(* IEC 61131-3 sources: TeoriaDeControl-NodeMCU/Lab2/build, 2 files *)

(* ---- plc.st ---- *)
TYPE
  LOGLEVEL : (CRITICAL, WARNING, INFO, DEBUG) := INFO;
END_TYPE

FUNCTION_BLOCK LOGGER
  VAR_INPUT
    TRIG : BOOL;
    MSG : STRING;
    LEVEL : LOGLEVEL := INFO;
  END_VAR
  VAR
    TRIG0 : BOOL;
  END_VAR

  IF TRIG AND NOT TRIG0 THEN
  {{
   LogMessage(GetFbVar(LEVEL),(char*)GetFbVar(MSG, .body),GetFbVar(MSG, .len));
  }}
  END_IF;
  TRIG0:=TRIG;
END_FUNCTION_BLOCK

FUNCTION_BLOCK python_eval
  VAR_INPUT
    TRIG : BOOL;
    CODE : STRING;
  END_VAR
  VAR_OUTPUT
    ACK : BOOL;
    RESULT : STRING;
  END_VAR
  VAR
    STATE : DWORD;
    BUFFER : STRING;
    PREBUFFER : STRING;
    TRIGM1 : BOOL;
    TRIGGED : BOOL;
  END_VAR

  {extern void __PythonEvalFB(int, PYTHON_EVAL*);__PythonEvalFB(0, data__);}
END_FUNCTION_BLOCK

FUNCTION_BLOCK python_poll
  VAR_INPUT
    TRIG : BOOL;
    CODE : STRING;
  END_VAR
  VAR_OUTPUT
    ACK : BOOL;
    RESULT : STRING;
  END_VAR
  VAR
    STATE : DWORD;
    BUFFER : STRING;
    PREBUFFER : STRING;
    TRIGM1 : BOOL;
    TRIGGED : BOOL;
  END_VAR

  {extern void __PythonEvalFB(int, PYTHON_EVAL*);__PythonEvalFB(1,(PYTHON_EVAL*)(void*)data__);}
END_FUNCTION_BLOCK

FUNCTION_BLOCK python_gear
  VAR_INPUT
    N : UINT;
    TRIG : BOOL;
    CODE : STRING;
  END_VAR
  VAR_OUTPUT
    ACK : BOOL;
    RESULT : STRING;
  END_VAR
  VAR
    py_eval : python_eval;
    COUNTER : UINT;
    _TMP_ADD10_OUT : UINT;
    _TMP_EQ13_OUT : BOOL;
    _TMP_SEL15_OUT : UINT;
    _TMP_AND7_OUT : BOOL;
  END_VAR

  _TMP_ADD10_OUT := ADD(COUNTER, 1);
  _TMP_EQ13_OUT := EQ(N, _TMP_ADD10_OUT);
  _TMP_SEL15_OUT := SEL(_TMP_EQ13_OUT, _TMP_ADD10_OUT, 0);
  COUNTER := _TMP_SEL15_OUT;
  _TMP_AND7_OUT := AND(_TMP_EQ13_OUT, TRIG);
  py_eval(TRIG := _TMP_AND7_OUT, CODE := CODE);
  ACK := py_eval.ACK;
  RESULT := py_eval.RESULT;
END_FUNCTION_BLOCK

PROGRAM Lab2
  VAR
    micro : INT;
    led1 : BOOL := 0;
    led2 : BOOL := 0;
    led3 : BOOL := 0;
    rele : BOOL := 0;
  END_VAR
  VAR
    TP1 : TP;
    TP2 : TP;
    TP3 : TP;
    TP4 : TP;
    _TMP_LE14_OUT : BOOL;
    _TMP_LE3_OUT : BOOL;
    _TMP_LE6_OUT : BOOL;
  END_VAR

  _TMP_LE14_OUT := LE(micro, 600);
  TP1(IN := _TMP_LE14_OUT, PT := T#10s);
  rele := TP1.Q;
  TP3(IN := _TMP_LE14_OUT, PT := T#3s);
  led3 := TP3.Q;
  _TMP_LE3_OUT := LE(micro, 800);
  TP2(IN := _TMP_LE3_OUT, PT := T#6s);
  led2 := TP2.Q;
  _TMP_LE6_OUT := LE(micro, 1000);
  TP4(IN := _TMP_LE6_OUT, PT := T#9s);
  led1 := TP4.Q;
END_PROGRAM

CONFIGURATION Config0

  RESOURCE Res0 ON PLC
    TASK task0(INTERVAL := T#20ms,PRIORITY := 0);
    PROGRAM instance0 WITH task0 : Lab2;
  END_RESOURCE
END_CONFIGURATION

(* ---- generated_plc.st ---- *)
PROGRAM Lab2
  VAR
    micro AT %IW0 : INT;
    led1 AT %QX0.1 : BOOL := 0;
    led2 AT %QX0.2 : BOOL := 0;
    led3 AT %QX0.3 : BOOL := 0;
    rele AT %QX0.0 : BOOL := 0;
  END_VAR
  VAR
    TP1 : TP;
    TP2 : TP;
    TP3 : TP;
    TP4 : TP;
    _TMP_LE14_OUT : BOOL;
    _TMP_LE3_OUT : BOOL;
    _TMP_LE6_OUT : BOOL;
  END_VAR

  _TMP_LE14_OUT := LE(micro, 600);
  TP1(IN := _TMP_LE14_OUT, PT := T#10s);
  rele := TP1.Q;
  TP3(IN := _TMP_LE14_OUT, PT := T#3s);
  led3 := TP3.Q;
  _TMP_LE3_OUT := LE(micro, 800);
  TP2(IN := _TMP_LE3_OUT, PT := T#6s);
  led2 := TP2.Q;
  _TMP_LE6_OUT := LE(micro, 1000);
  TP4(IN := _TMP_LE6_OUT, PT := T#9s);
  led1 := TP4.Q;
END_PROGRAM

CONFIGURATION Config0

  RESOURCE Res0 ON PLC
    TASK task0(INTERVAL := T#20ms,PRIORITY := 0);
    PROGRAM instance0 WITH task0 : Lab2;
  END_RESOURCE
END_CONFIGURATION
